// TIA Portal V16 export
// export: Created 2021-07-12T14:47:18.5347053Z, ExportSetting WithDefaults, DisplayName Totally Integrated Automation Portal, DisplayVersion V16, DisplayName TIA Portal Version Control Interface, DisplayVersion V16, DisplayName TIA Portal Openness, DisplayVersion V16, DisplayName STEP 7 Professional, DisplayVersion V16, DisplayName STEP 7 Safety, DisplayVersion V16, DisplayName WinCC Professional, DisplayVersion V16
TYPE "SimaHydTO_typeIHMIConnectionBasicAxisControlDirectOutput"
TITLE = SimaHydTO_typeIHMIConnectionBasicAxisControlDirectOutput
// Direct output control
// stored: IsFailsafeCompliant false
   STRUCT
      jogForward : Bool;   // Direct output is active in positive direction if TRUE
      jogBackward : Bool;   // Direct output is active in negative direction if TRUE
      commandValueForward : LReal := 5.0;   // Direct output value in positive direction [%]
      commandValueBackward : LReal := 5.0;   // Direct output value in negative direction [%]
      commandValueRamp : LReal := 100.0;   // Ramp for command value [%/s]
      safetyDistance : LReal := 50.0;   // Safety distance to avoid passing over the min. and max. positions
   END_STRUCT;
END_TYPE
